ABB RAPID module: GoHome.mod

MODULE GoHome
    CONST robtarget Target_10:=[[-59.887841644,22.215507517,-50.081855147],[0.707106781,0.00000082,-0.00000082,-0.707106781],[0,0,0,1],[9E+09,9E+09,9E+09,9E+09,9E+09,9E+09]];
    CONST robtarget Target_20:=[[-59.887957505,22.215507517,-0.081855147],[0.707106781,0.00000082,-0.00000082,-0.707106781],[0,0,0,1],[9E+09,9E+09,9E+09,9E+09,9E+09,9E+09]];
    CONST robtarget Target_30:=[[-59.887957505,38.001461443,-0.081855147],[0.707106781,0.00000082,-0.00000082,-0.707106781],[0,0,0,1],[9E+09,9E+09,9E+09,9E+09,9E+09,9E+09]];
    CONST robtarget Target_40:=[[-93.271368484,38.001461443,-0.081932504],[0.707106781,0.000000819,-0.000000819,-0.707106781],[0,0,0,1],[9E+09,9E+09,9E+09,9E+09,9E+09,9E+09]];
    CONST robtarget Target_50:=[[-100.93542349,34.650363976,-0.081950263],[0.707106781,0.00000082,-0.000000819,-0.707106781],[0,0,0,1],[9E+09,9E+09,9E+09,9E+09,9E+09,9E+09]];
    CONST robtarget Target_60:=[[-103.679130867,26.748486782,-0.081956621],[0.707106782,0.00000082,-0.000000819,-0.707106781],[0,0,0,1],[9E+09,9E+09,9E+09,9E+09,9E+09,9E+09]];
    CONST robtarget Target_70:=[[-99.741021774,19.368860088,-0.081947494],[0.707106781,0.000000819,-0.00000082,-0.707106781],[0,0,0,1],[9E+09,9E+09,9E+09,9E+09,9E+09,9E+09]];
    CONST robtarget Target_80:=[[-99.740905914,19.368860088,-50.081947495],[0.707106781,0.000000819,-0.00000082,-0.707106781],[0,0,0,1],[9E+09,9E+09,9E+09,9E+09,9E+09,9E+09]];
    CONST robtarget Target_90:=[[-59.88784141,49.388051159,-50.081855147],[0.707106781,0.00000082,-0.00000082,-0.707106781],[0,0,0,1],[9E+09,9E+09,9E+09,9E+09,9E+09,9E+09]];
    CONST robtarget Target_100:=[[-59.887957271,49.388051159,-0.081855147],[0.707106781,0.00000082,-0.00000082,-0.707106781],[0,0,0,1],[9E+09,9E+09,9E+09,9E+09,9E+09,9E+09]];
    CONST robtarget Target_110:=[[-61.656166444,68.408831548,-0.081859245],[0.707106782,0.00000082,-0.000000819,-0.707106781],[0,0,0,1],[9E+09,9E+09,9E+09,9E+09,9E+09,9E+09]];
    CONST robtarget Target_120:=[[-73.086050217,75.007878021,-0.08188573],[0.707106781,0.000000819,-0.000000819,-0.707106781],[0,0,0,1],[9E+09,9E+09,9E+09,9E+09,9E+09,9E+09]];
    CONST robtarget Target_130:=[[-93.012582397,73.204998124,-0.081931904],[0.707106781,0.000000819,-0.000000819,-0.707106781],[0,0,0,1],[9E+09,9E+09,9E+09,9E+09,9E+09,9E+09]];
    CONST robtarget Target_140:=[[-99.741021774,61.550999266,-0.081947494],[0.707106781,0.00000082,-0.00000082,-0.707106781],[0,0,0,1],[9E+09,9E+09,9E+09,9E+09,9E+09,9E+09]];
    CONST robtarget Target_150:=[[-99.741021774,49.388051159,-0.081947494],[0.707106781,0.00000082,-0.00000082,-0.707106781],[0,0,0,1],[9E+09,9E+09,9E+09,9E+09,9E+09,9E+09]];
    CONST robtarget Target_160:=[[-59.887957271,49.388051159,-0.081855147],[0.707106781,0.000000819,-0.000000819,-0.707106781],[0,0,0,1],[9E+09,9E+09,9E+09,9E+09,9E+09,9E+09]];
    CONST robtarget Target_170:=[[-59.88784141,49.388051159,-50.081855147],[0.707106781,0.000000819,-0.000000819,-0.707106781],[0,0,0,1],[9E+09,9E+09,9E+09,9E+09,9E+09,9E+09]];
    CONST robtarget Target_180:=[[-59.88784141,111.75550847,-50.081855147],[0.707106781,0.00000082,-0.00000082,-0.707106781],[0,0,0,1],[9E+09,9E+09,9E+09,9E+09,9E+09,9E+09]];
    CONST robtarget Target_190:=[[-59.887957271,111.75550847,-0.081855147],[0.707106781,0.00000082,-0.00000082,-0.707106781],[0,0,0,1],[9E+09,9E+09,9E+09,9E+09,9E+09,9E+09]];
    CONST robtarget Target_200:=[[-61.656166444,130.776288859,-0.081859245],[0.707106782,0.00000082,-0.000000819,-0.707106781],[0,0,0,1],[9E+09,9E+09,9E+09,9E+09,9E+09,9E+09]];
    CONST robtarget Target_210:=[[-73.086050217,137.375335333,-0.08188573],[0.707106781,0.000000819,-0.000000819,-0.707106781],[0,0,0,1],[9E+09,9E+09,9E+09,9E+09,9E+09,9E+09]];
    CONST robtarget Target_220:=[[-93.012582397,135.572455435,-0.081931904],[0.707106781,0.000000819,-0.000000819,-0.707106781],[0,0,0,1],[9E+09,9E+09,9E+09,9E+09,9E+09,9E+09]];
    CONST robtarget Target_230:=[[-99.741021774,123.918456577,-0.081947494],[0.707106781,0.00000082,-0.00000082,-0.707106781],[0,0,0,1],[9E+09,9E+09,9E+09,9E+09,9E+09,9E+09]];
    CONST robtarget Target_240:=[[-99.741021774,111.75550847,-0.081947494],[0.707106781,0.00000082,-0.00000082,-0.707106781],[0,0,0,1],[9E+09,9E+09,9E+09,9E+09,9E+09,9E+09]];
    CONST robtarget Target_250:=[[-59.887957271,111.75550847,-0.081855147],[0.707106781,0.000000819,-0.000000819,-0.707106781],[0,0,0,1],[9E+09,9E+09,9E+09,9E+09,9E+09,9E+09]];
    CONST robtarget Target_260:=[[-59.88784141,111.75550847,-50.081855147],[0.707106781,0.000000819,-0.000000819,-0.707106781],[0,0,0,1],[9E+09,9E+09,9E+09,9E+09,9E+09,9E+09]];
    CONST robtarget Target_270:=[[-99.740905914,144.97534301,-50.081947495],[0.707106781,0.000000819,-0.000000819,-0.707106781],[0,0,0,1],[9E+09,9E+09,9E+09,9E+09,9E+09,9E+09]];
    CONST robtarget Target_280:=[[-99.741021774,144.97534301,-0.081947494],[0.707106781,0.000000819,-0.000000819,-0.707106781],[0,0,0,1],[9E+09,9E+09,9E+09,9E+09,9E+09,9E+09]];
    CONST robtarget Target_290:=[[-59.983167415,144.97534301,-0.081855368],[0.707106781,0.000000819,-0.000000819,-0.707106781],[0,0,0,1],[9E+09,9E+09,9E+09,9E+09,9E+09,9E+09]];
    CONST robtarget Target_300:=[[-59.983167415,157.043081207,-0.081855368],[0.707106781,0.00000082,-0.00000082,-0.707106781],[0,0,0,1],[9E+09,9E+09,9E+09,9E+09,9E+09,9E+09]];
    CONST robtarget Target_310:=[[-66.114081356,167.662135648,-0.081869575],[0.707106781,0.000000819,-0.000000819,-0.707106781],[0,0,0,1],[9E+09,9E+09,9E+09,9E+09,9E+09,9E+09]];
    CONST robtarget Target_320:=[[-78.375909236,167.662135648,-0.081897988],[0.707106781,0.000000819,-0.000000819,-0.707106781],[0,0,0,1],[9E+09,9E+09,9E+09,9E+09,9E+09,9E+09]];
    CONST robtarget Target_330:=[[-84.506823176,151.009212109,-0.081912194],[0.707106781,0.00000082,-0.00000082,-0.707106781],[0,0,0,1],[9E+09,9E+09,9E+09,9E+09,9E+09,9E+09]];
    CONST robtarget Target_340:=[[-84.506707316,151.009212109,-50.081912194],[0.707106781,0.00000082,-0.00000082,-0.707106781],[0,0,0,1],[9E+09,9E+09,9E+09,9E+09,9E+09,9E+09]];
    CONST robtarget Target_350:=[[-145.225874554,122.068654602,-50.082052893],[0.707106781,0.000000819,-0.000000819,-0.707106781],[-1,-1,0,1],[9E+09,9E+09,9E+09,9E+09,9E+09,9E+09]];
    CONST robtarget Target_360:=[[-145.225990414,122.068654602,-0.082052893],[0.707106781,0.000000819,-0.000000819,-0.707106781],[0,0,0,1],[9E+09,9E+09,9E+09,9E+09,9E+09,9E+09]];
    CONST robtarget Target_370:=[[-216.314272977,130.011265242,-0.08221762],[0.707106782,0.00000082,-0.000000819,-0.707106781],[-1,-1,0,1],[9E+09,9E+09,9E+09,9E+09,9E+09,9E+09]];
    CONST robtarget Target_380:=[[-238.920712,122.070831135,-0.082270004],[0.707106781,0.00000082,-0.00000082,-0.707106781],[-1,-1,0,1],[9E+09,9E+09,9E+09,9E+09,9E+09,9E+09]];
    CONST robtarget Target_390:=[[-242.176963668,87.21495429,-0.082277549],[0.707106781,0.000000819,-0.000000819,-0.707106781],[-1,-1,0,1],[9E+09,9E+09,9E+09,9E+09,9E+09,9E+09]];
    CONST robtarget Target_400:=[[-235.683786475,78.752058887,-0.082262503],[0.707106781,0.000000819,-0.000000819,-0.707106781],[-1,-1,0,1],[9E+09,9E+09,9E+09,9E+09,9E+09,9E+09]];
    CONST robtarget Target_410:=[[-228.457991082,81.055519424,-0.082245759],[0.707106781,0.000000819,-0.000000819,-0.707106781],[-1,-1,0,1],[9E+09,9E+09,9E+09,9E+09,9E+09,9E+09]];
    CONST robtarget Target_420:=[[-223.813275477,95.060731266,-0.082234996],[0.707106781,0.000000819,-0.000000819,-0.707106781],[-1,-1,0,1],[9E+09,9E+09,9E+09,9E+09,9E+09,9E+09]];
    CONST robtarget Target_430:=[[-205.993838978,96.347520237,-0.082193705],[0.707106781,0.000000819,-0.00000082,-0.707106782],[-1,-1,0,1],[9E+09,9E+09,9E+09,9E+09,9E+09,9E+09]];
    CONST robtarget Target_440:=[[-207.00309405,72.842237427,-0.082196044],[0.707106782,0.000000819,-0.000000818,-0.707106781],[-1,-1,0,1],[9E+09,9E+09,9E+09,9E+09,9E+09,9E+09]];
    CONST robtarget Target_450:=[[-227.772910705,70.716966245,-0.082244172],[0.707106781,0.000000819,-0.000000819,-0.707106781],[-1,-1,0,1],[9E+09,9E+09,9E+09,9E+09,9E+09,9E+09]];
    CONST robtarget Target_460:=[[-231.882732587,35.693817055,-0.082253695],[0.707106781,0.000000819,-0.000000819,-0.707106781],[-1,-1,0,1],[9E+09,9E+09,9E+09,9E+09,9E+09,9E+09]];
    CONST robtarget Target_470:=[[-225.128328942,25.434710387,-0.082238044],[0.707106781,0.000000819,-0.000000819,-0.707106781],[-1,-1,0,1],[9E+09,9E+09,9E+09,9E+09,9E+09,9E+09]];
    CONST robtarget Target_480:=[[-215.976129925,26.869358271,-0.082216836],[0.707106781,0.00000082,-0.00000082,-0.707106781],[-1,-1,0,1],[9E+09,9E+09,9E+09,9E+09,9E+09,9E+09]];
    CONST robtarget Target_490:=[[-212.521294514,45.774375392,-0.08220883],[0.707106781,0.000000819,-0.000000819,-0.707106781],[-1,-1,0,1],[9E+09,9E+09,9E+09,9E+09,9E+09,9E+09]];
    CONST robtarget Target_500:=[[-132.204623558,69.10534384,-0.08202272],[0.707106781,0.000000819,-0.00000082,-0.707106782],[0,0,0,1],[9E+09,9E+09,9E+09,9E+09,9E+09,9E+09]];
    CONST robtarget Target_510:=[[-131.099190925,103.471454414,-0.082020159],[0.707106781,0.000000819,-0.000000819,-0.707106781],[0,0,0,1],[9E+09,9E+09,9E+09,9E+09,9E+09,9E+09]];
    CONST robtarget Target_520:=[[-145.225990414,122.068654602,-0.082052893],[0.707106781,0.000000819,-0.000000819,-0.707106781],[0,0,0,1],[9E+09,9E+09,9E+09,9E+09,9E+09,9E+09]];
    CONST robtarget Target_530:=[[-145.225874554,122.068654602,-50.082052893],[0.707106781,0.000000819,-0.000000819,-0.707106781],[-1,-1,0,1],[9E+09,9E+09,9E+09,9E+09,9E+09,9E+09]];
    CONST robtarget Target_540:=[[-143.491221184,87.474940519,-50.082048873],[0.707106781,0.000000819,-0.000000819,-0.707106781],[-1,-1,0,1],[9E+09,9E+09,9E+09,9E+09,9E+09,9E+09]];
    CONST robtarget Target_550:=[[-143.491337044,87.474940519,-0.082048874],[0.707106781,0.000000819,-0.000000819,-0.707106781],[0,0,0,1],[9E+09,9E+09,9E+09,9E+09,9E+09,9E+09]];
    CONST robtarget Target_560:=[[-145.497156615,75.291484437,-0.082053521],[0.707106781,0.000000819,-0.000000819,-0.707106781],[0,0,0,1],[9E+09,9E+09,9E+09,9E+09,9E+09,9E+09]];
    CONST robtarget Target_570:=[[-153.701887033,72.48506132,-0.082072534],[0.707106781,0.000000819,-0.00000082,-0.707106782],[0,0,0,1],[9E+09,9E+09,9E+09,9E+09,9E+09,9E+09]];
    CONST robtarget Target_580:=[[-160.745274412,94.690565784,-0.082088855],[0.707106782,0.00000082,-0.000000819,-0.707106781],[0,0,0,1],[9E+09,9E+09,9E+09,9E+09,9E+09,9E+09]];
    CONST robtarget Target_590:=[[-157.752837767,106.504530415,-0.082081921],[0.707106782,0.000000819,-0.000000818,-0.707106781],[0,0,0,1],[9E+09,9E+09,9E+09,9E+09,9E+09,9E+09]];
    CONST robtarget Target_600:=[[-150.089305159,109.52469583,-0.082064163],[0.707106781,0.000000819,-0.000000819,-0.707106781],[0,0,0,1],[9E+09,9E+09,9E+09,9E+09,9E+09,9E+09]];
    CONST robtarget Target_610:=[[-143.491337044,87.474940519,-0.082048874],[0.707106781,0.000000819,-0.000000819,-0.707106781],[0,0,0,1],[9E+09,9E+09,9E+09,9E+09,9E+09,9E+09]];
    CONST robtarget Target_620:=[[-143.491221184,87.474940519,-50.082048873],[0.707106781,0.000000819,-0.000000819,-0.707106781],[-1,-1,0,1],[9E+09,9E+09,9E+09,9E+09,9E+09,9E+09]];
    CONST robtarget MidPoint:=[[81.533842296,132.215507517,-191.502883681],[0.707106781,0.00000082,-0.00000082,-0.707106781],[0,-2,-2,0],[9E+09,9E+09,9E+09,9E+09,9E+09,9E+09]];
    CONST jointtarget Home:=[[0,0,0,0,0,0],[9E+09,9E+09,9E+09,9E+09,9E+09,9E+09]];
    CONST jointtarget PosMant:=[[-28,50,-40,0,-20,0],[9E+09,9E+09,9E+09,9E+09,9E+09,9E+09]];
ENDMODULE
